INTERFACE I_Fault

METHOD Acknowledge
VAR_INPUT
END_VAR
END_METHOD

METHOD Clear
VAR_INPUT
END_VAR
END_METHOD

PROPERTY FaultCode : UDINT
GET
END_GET
END_PROPERTY

PROPERTY FaultMessage : STRING
GET
END_GET
END_PROPERTY

PROPERTY IsAcknowledged : BOOL
GET
END_GET
END_PROPERTY

PROPERTY IsActive : BOOL
GET
END_GET
END_PROPERTY

METHOD Raise
VAR_INPUT
END_VAR
END_METHOD

PROPERTY Severity : E_FaultSeverity
GET
END_GET
END_PROPERTY

PROPERTY Timestamp : DATE_AND_TIME
GET
END_GET
END_PROPERTY

END_INTERFACE

(* stored: Version 1.1.0.1, ProductVersion 3.1.4026.18
   Itf I_Fault: Id {3d7523ee-f469-41b2-95c2-31b6dda08954}
   Method Acknowledge: Id {5a46c8ca-17a6-4f6e-a036-a1b00313fd52}
   Method Clear: Id {0b1a43e6-4315-4e36-8da0-333b4ff3d02c}
   Property FaultCode: Id {73d32827-1592-4f08-9334-f1c19d70846f}
   Get Get: Id {3e95e720-a472-45df-ad72-25aab5eb4b09}
   Property FaultMessage: Id {faefed8a-e0b8-4d48-98c9-5bd76316d570}
   Get Get: Id {ccdc0936-2405-4a96-945b-3fbd8806a8a7}
   Property IsAcknowledged: Id {4fb3a720-70d9-4d1f-86fe-9958ca79b602}
   Get Get: Id {da348f12-8977-4e36-9287-5f92446d58ad}
   Property IsActive: Id {19632952-32e7-4d15-ba42-557b94624653}
   Get Get: Id {a2b608ca-b008-440c-bf85-7d24cb080774}
   Method Raise: Id {8a0336eb-8fd1-4e6c-b812-8a1106f335d2}
   Property Severity: Id {9e30a77b-2f79-4a27-9e00-2d1e9b8d03f5}
   Get Get: Id {12f48f59-2eaf-4bd7-9dd0-833df7d7750c}
   Property Timestamp: Id {d35243b6-5811-479e-8960-5df9c7f4968c}
   Get Get: Id {62bada3c-464d-457e-a748-11a7bec29dff} *)
